// TIA Portal V21 export
// export: Created 2026-05-11T00:00:00.0000000Z, ExportSetting None, DisplayName Totally Integrated Automation Portal, DisplayVersion V21, DisplayName STEP 7 Professional, DisplayVersion V21
FUNCTION "MCPVerify_FC_LAD" : Void   // FC901, LAD
TITLE = MCP LAD 原生指令验证
{ S7_Optimized_Access := 'TRUE' }
// MCP 验证：LAD 原生指令 6 网络（串联/并联/SR/比较/Move/Add）
// stored: AutoNumber false, SetENOAutomatically false
   VAR_INPUT
      "A" : Bool;
      "B" : Bool;
      SET : Bool;
      RESET : Bool;
      V1 : Int;
      V2 : Int;
      VAL : Int;
   END_VAR
   VAR_OUTPUT
      OUT_AND : Bool;
      OUT_OR : Bool;
      OUT_SR : Bool;
      OUT_GT : Bool;
      DST : Int;
      SUM : Int;
   END_VAR
BEGIN

REGION Network 1: N1-串联
   // 串联 AND：A & B -> OUT_AND
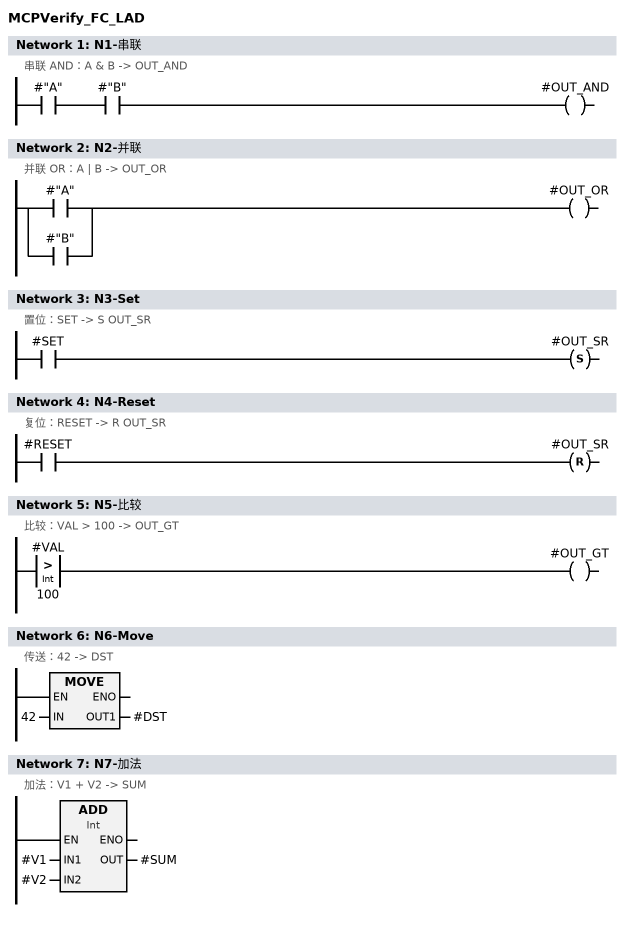
   RUNG wire#powerrail
      Contact( #"A" )
      Contact( #"B" )
      Coil( #OUT_AND )
   END_RUNG
   // the same network as SCL:
   #OUT_AND := #"A" AND #"B";
END_REGION

REGION Network 2: N2-并联
   // 并联 OR：A | B -> OUT_OR
   RUNG wire#powerrail
      Contact( #"A" )
      wire#w1
      Coil( #OUT_OR )
   END_RUNG
   RUNG wire#powerrail
      Contact( #"B" )
   END_RUNG wire#w1
   // the same network as SCL:
   #OUT_OR := #"A" OR #"B";
END_REGION

REGION Network 3: N3-Set
   // 置位：SET -> S OUT_SR
   RUNG wire#powerrail
      Contact( #SET )
      S_Coil( #OUT_SR )
   END_RUNG
   // the same network as SCL:
   IF #SET THEN #OUT_SR := TRUE; END_IF;
END_REGION

REGION Network 4: N4-Reset
   // 复位：RESET -> R OUT_SR
   RUNG wire#powerrail
      Contact( #RESET )
      R_Coil( #OUT_SR )
   END_RUNG
   // the same network as SCL:
   IF #RESET THEN #OUT_SR := FALSE; END_IF;
END_REGION

REGION Network 5: N5-比较
   // 比较：VAL > 100 -> OUT_GT
   RUNG wire#powerrail
      { S7_Templates := "SrcType := Int" } GT_Contact(in1 := #VAL, in2 := 100)
      Coil( #OUT_GT )
   END_RUNG
   // the same network as SCL:
   #OUT_GT := #VAL > 100;
END_REGION

REGION Network 6: N6-Move
   // 传送：42 -> DST
   RUNG wire#powerrail
      Move(in := 42, out1 => #DST)
   END_RUNG
   // the same network as SCL:
   #DST := 42;
END_REGION

REGION Network 7: N7-加法
   // 加法：V1 + V2 -> SUM
   RUNG wire#powerrail
      { S7_Templates := "SrcType := Int" } Add(in1 := #V1, in2 := #V2, out => #SUM)
   END_RUNG
   // the same network as SCL:
   #SUM := #V1 + #V2;
END_REGION
END_FUNCTION
